FUNCTION_BLOCK FB_TestSuite1 EXTENDS FB_TestSuite
VAR_INPUT
END_VAR
VAR_OUTPUT
END_VAR
VAR
END_VAR

TestCase1A();
TestCase1BCD();
TestCase1F_IgnoreCase();

METHOD TestCase1BCD
VAR_INPUT
END_VAR
TEST('TestCase1B');

AssertTrue(False, 'Condition is not true');

TEST_FINISHED_NAMED('TestCase1B');

IF TEST_ORDERED('TestCase1C') THEN

    AssertTrue(TRUE, 'Condition is not true');

    TEST_FINISHED();
END_IF

TEST('TestCase1D');

AssertTrue(FALSE, 'Condition is not true');
AssertTrue(TRUE, 'Condition is not true');


TEST_FINISHED();


TEST('TestCase1E with a space');

AssertTrue(TRUE, 'Condition is not true');
AssertTrue(TRUE, 'Condition is not true');


TEST_FINISHED();
END_METHOD

METHOD TestCase1F_IgnoreCase : REFERENCE TO FB_Test
VAR_INPUT
END_VAR
VAR_INST
    step : DINT;
END_VAR

IF TesT_ORdEReD('TestCase1F Ignore Case') THEN
    AssertFalse(False, 'Condition is not false');
    // introduce whitespace for test        
            TEsT_FiNiSHED();
END_IF
END_METHOD

METHOD TestCase1A
VAR_INPUT
END_VAR
TEST('TestCase1A');

AssertTrue(2+2=4, 'Condition is not true');

TEST_FINISHED();
END_METHOD

END_FUNCTION_BLOCK

(* stored: Version 1.1.0.1, ProductVersion 3.1.4024.12
   POU FB_TestSuite1: Id {a5ea8811-5301-4f6c-aafd-b2e96e83b4a4}, SpecialFunc None
   Method TestCase1BCD: Id {5dcda336-eb7c-4bc2-a049-4f178c78790e}
   Method TestCase1F_IgnoreCase: Id {93ccc455-0496-40f6-9dd8-d004dfed4904}
   Method TestCase1A: Id {976e0437-3cd7-4f7e-af64-671bf9c25b18} *)
